TYPE ST_GeneralAlarm :
STRUCT
	bEmergencyStopActive : BOOL := FALSE; // Alarm status active
	bSystemFault         : BOOL := FALSE; // General system failure
	sMessage             : STRING(80) := ''; // General alarm message
END_STRUCT
END_TYPE

(* stored: Version 1.1.0.1, ProductVersion 3.1.4024.12
   DUT ST_GeneralAlarm: Id {31799fea-0f46-44aa-ab45-e8ff88c72765} *)
